TYPE MachineComRequest :
STRUCT
  Start : BOOL;
  Stop : BOOL;
  GoHome : BOOL;
  Halt : BOOL;
END_STRUCT
END_TYPE

(* stored: Version 1.1.0.1
   DUT MachineComRequest: Id {ca4e739a-0473-4c05-bd3e-49b0920a09f2} *)
